FUNCTION_BLOCK Interpolate
VAR_INPUT
	EN: BOOL;
	x: LREAL;
END_VAR
VAR_OUTPUT
	ENO: BOOL;
	y: LREAL;
END_VAR
VAR CONSTANT
	NUM_POINTS: INT := 9;
END_VAR
VAR
	i: INT;
	j: INT;
	ss: LREAL;
	t: LREAL;
	k: LREAL;
END_VAR
VAR PERSISTENT
	xd: ARRAY [0..NUM_POINTS - 1] OF LREAL;
	yd: ARRAY [0..NUM_POINTS - 1] OF LREAL;
END_VAR

ENO := EN;
k := 0;
FOR i := 0 TO NUM_POINTS - 1 DO
	ss := 1;
	t := 1;
	FOR j := 0 TO NUM_POINTS - 1 DO
		IF i <> j THEN			
			ss := ss * (x - xd[j]);
			t := t * (xd[i] - xd[j]);
		END_IF
	END_FOR
	IF t <> 0 THEN
		k := k + ((ss / t) * yd[i]);		
	END_IF
END_FOR
y := k;

END_FUNCTION_BLOCK

(* stored: Version 1.1.0.1, ProductVersion 3.1.4024.3
   POU Interpolate: Id {0c7a3a39-b100-4547-a3f5-05d6cc77f908}, SpecialFunc None *)
